FUNCTION_BLOCK FB_Queue_Stack IMPLEMENTS I_Stack
VAR_INPUT
END_VAR
VAR_OUTPUT
END_VAR
VAR
END_VAR

{warning 'add method implementation '}
METHOD Peek : T_DATA_TYPE
END_METHOD

{warning 'add method implementation '}
METHOD Pop
END_METHOD

{warning 'add method implementation '}
METHOD Push
VAR_INPUT
	Data	: T_DATA_TYPE;
END_VAR
END_METHOD

{warning 'add method implementation '}
METHOD Show
END_METHOD

END_FUNCTION_BLOCK

(* stored: Version 1.1.0.1, ProductVersion 3.1.4024.4
   POU FB_Queue_Stack: Id {f248fb0a-d0a2-4ad6-84b3-ed190aee8290}, SpecialFunc None
   Method Peek: Id {18190e9c-a2e4-4e82-bd24-c801e3a00d7a}
   Method Pop: Id {c4574ff8-375c-4b2c-85f4-890732572ca9}
   Method Push: Id {90e5158c-1a1a-4bbe-9c95-68066520ce31}
   Method Show: Id {13d89b5a-ee98-40b0-9f4b-68da6cae9832} *)
